FUNCTION_BLOCK FB_Abfullmodul
VAR_INPUT
    bEnable: BOOL;
    bExecute : BOOL;
END_VAR
VAR_OUTPUT
    eState : eBetriebszustand;
END_VAR
VAR
    nState : INT := 0;
    nStation :INT := 0;
    
    fbVereinzelung : FB_Vereinzelung;
    fbTransport : FB_Transport;
    fbDispenser1 : FB_Dispenser;
    fbDispenser2 : FB_Dispenser;
    fbDispenser3 : FB_Dispenser;
	fbEZylinder1: FB_EZylinder;
	fbEZylinder2: FB_EZylinder;
END_VAR
VAR_IN_OUT
    ax1 : AXIS_REF;
	ax2 : AXIS_REF;
	ax3 : AXIS_REF;
END_VAR

fbVereinzelung(
	bEnable:= bEnable, 
	bExecute:= , 
	bSensor1:= IFC_HW.bEinzelSens1, 
	bSensor2:= IFC_HW.bEinzelSens2, 
	bSensor3:= IFC_HW.bEinzelSens3, 
	bSensor4:= IFC_HW.bBandSens1, 
	eState=> , 
	bGate1=> fbEZylinder1.bGate, 
	bGate2=> fbEZylinder2.bGate);
	
fbEZylinder1(bGate:= , bError:= , bR1=> IFC_HW.bR1AKT1, bR2=> IFC_HW.bR2AKT1);
fbEZylinder2(bGate:= , bError:= , bR1=> IFC_HW.bR1AKT2, bR2=> IFC_HW.bR2AKT2);

fbTransport(
	bEnable:= bEnable, 
	bExecute:= , 
	nStation:= nStation, 
	bSens1:= IFC_HW.bBandSens1, 
	bSens2:= IFC_HW.bBandSens2, 
	bSens3:= IFC_HW.bBandSens3, 
	bSens4:= IFC_HW.bBandSens4, 
	eState=> , 
	bStopper1=> IFC_HW.bBandHub1, 
	bStopper2=> IFC_HW.bBandHub2, 
	bStopper3=> IFC_HW.bBandHub3, 
	ax:= IFC_HW.ax_BandMotor);
	
fbDispenser1(
	bEnable:= bEnable, 
	bExecute:= , 
	rDistance:= 100, 
	eState=> , 
	ax:= ax1);

fbDispenser2(
	bEnable:= bEnable, 
	bExecute:= , 
	rDistance:= 100, 
	eState=> , 
	ax:= ax2);

fbDispenser3(
	bEnable:= bEnable, 
	bExecute:= , 
	rDistance:= 100, 
	eState=> , 
	ax:= ax3);

CASE nState OF
	
	0: // OFF
	eState := eBetriebszustand.OFF;
	
	fbVereinzelung.bEnable := FALSE;
	fbTransport.bEnable := FALSE;
	fbDispenser1.bEnable := FALSE;
	fbDispenser2.bEnable := FALSE;
	fbDispenser3.bEnable := FALSE;
	
	fbVereinzelung.bExecute := FALSE;
	fbTransport.bExecute := FALSE;
	fbDispenser1.bExecute := FALSE;
	fbDispenser2.bExecute := FALSE;
	fbDispenser3.bExecute := FALSE;
	
	IF bEnable THEN
		nState:= 10; // INIT
	END_IF
	
	10: // INIT
	eState := eBetriebszustand.INIT;
	
	fbVereinzelung.bEnable := TRUE;
	fbTransport.bEnable := TRUE;
	fbDispenser1.bEnable := TRUE;
	fbDispenser2.bEnable := TRUE;
	fbDispenser3.bEnable := TRUE;
	
	fbVereinzelung.bExecute := FALSE;
	fbTransport.bExecute := FALSE;
	fbDispenser1.bExecute := FALSE;
	fbDispenser2.bExecute := FALSE;
	fbDispenser3.bExecute := FALSE;
	
	IF (fbVereinzelung.eState = eBetriebszustand.READY) AND (fbTransport.eState = eBetriebszustand.READY) AND (fbDispenser1.eState = eBetriebszustand.READY) 
		AND (fbDispenser2.eState = eBetriebszustand.READY) AND (fbDispenser3.eState = eBetriebszustand.READY) THEN
		
		nState := 20; // READY
	END_IF
	
	20: // READY
	eState := eBetriebszustand.READY;
	
	fbVereinzelung.bEnable := TRUE;
	fbTransport.bEnable := TRUE;
	fbDispenser1.bEnable := TRUE;
	fbDispenser2.bEnable := TRUE;
	fbDispenser3.bEnable := TRUE;
	
	IF bExecute THEN
		nState := 30; //Start
	END_IF
	
	30: // PROD - Start
	eState := eBetriebszustand.PROD;
	nStation := 1;
	
	fbVereinzelung.bEnable := TRUE;
	fbTransport.bEnable := TRUE;
	fbDispenser1.bEnable := TRUE;
	fbDispenser2.bEnable := TRUE;
	fbDispenser3.bEnable := TRUE;
	
	fbVereinzelung.bExecute := TRUE;
	fbTransport.bExecute := TRUE;
	fbDispenser1.bExecute := FALSE;
	fbDispenser2.bExecute := FALSE;
	fbDispenser3.bExecute := FALSE;
	
	IF (fbVereinzelung.eState = eBetriebszustand.DONE) AND (fbTransport.eState = eBetriebszustand.DONE)THEN
		nState := 31; // Extruder 1
	END_IF
	
	31: // PROD - Extruder 1
	eState := eBetriebszustand.PROD;
	nStation := 1;

	fbVereinzelung.bExecute := FALSE;
	fbTransport.bExecute := FALSE;
	fbDispenser1.bExecute := TRUE;
	fbDispenser2.bExecute := FALSE;
	fbDispenser3.bExecute := FALSE;
	
	IF fbDispenser1.eState = eBetriebszustand.DONE THEN
		nState := 32; // Bewegung zu Station 2
	END_IF
	
	32: // PROD - Bewegung zu Station 2
	eState := eBetriebszustand.PROD;
	nStation := 2;
	
	fbVereinzelung.bExecute := FALSE;
	fbTransport.bExecute := TRUE;
	fbDispenser1.bExecute := FALSE;
	fbDispenser2.bExecute := FALSE;
	fbDispenser3.bExecute := FALSE;
	
	IF fbTransport.eState = eBetriebszustand.DONE THEN
		nState := 33; //  Extruder 2
	END_IF
	
	33: // PROD - Extruder 2
	eState := eBetriebszustand.PROD;
	nStation := 2;
	
	fbVereinzelung.bExecute := FALSE;
	fbTransport.bExecute := FALSE;
	fbDispenser1.bExecute := FALSE;
	fbDispenser2.bExecute := TRUE;
	fbDispenser3.bExecute := FALSE;
	
	IF fbDispenser2.eState = eBetriebszustand.DONE THEN
		nState := 34; // Bewegung zu Station 3
	END_IF
	
	34: // PROD - Bewegung zu Station 3
	eState := eBetriebszustand.PROD;
	nStation := 3;
	
	fbVereinzelung.bExecute := FALSE;
	fbTransport.bExecute := TRUE;
	fbDispenser1.bExecute := FALSE;
	fbDispenser2.bExecute := FALSE;
	fbDispenser3.bExecute := FALSE;
	
	IF fbTransport.eState = eBetriebszustand.DONE THEN
		nState := 35; // Extruder 3
	END_IF
	
	35: // PROD - Extruder 3
	eState := eBetriebszustand.PROD;
	nStation := 3;
	
	fbVereinzelung.bExecute := FALSE;
	fbTransport.bExecute := FALSE;
	fbDispenser1.bExecute := FALSE;
	fbDispenser2.bExecute := FALSE;
	fbDispenser3.bExecute := TRUE;
	
	IF fbDispenser3.eState = eBetriebszustand.DONE THEN
		nState := 36; // Bewegung zu Abholstation
	END_IF
	
	36: // PROD - Bewegung zu Abholstation
	eState := eBetriebszustand.PROD;
	nStation := 4;
	
	fbVereinzelung.bExecute := FALSE;
	fbTransport.bExecute := TRUE;
	fbDispenser1.bExecute := FALSE;
	fbDispenser2.bExecute := FALSE;
	fbDispenser3.bExecute := FALSE; 
	
	IF fbTransport.eState = eBetriebszustand.DONE THEN
		nState := 40; // DONE
	END_IF
	
	40: // DONE
	eState :=  eBetriebszustand.DONE;
	nStation := 4;
	
	IF NOT bExecute THEN
		nState := 20; // READY
	ELSIF nStation = 4 THEN
		nState := 30; // START
	END_IF
	
END_CASE

END_FUNCTION_BLOCK

(* stored: Version 1.1.0.1, ProductVersion 3.1.4024.15
   POU FB_Abfullmodul: Id {0d4ac5ca-edd1-416b-acfb-b45ddda04365}, SpecialFunc None *)
